Fanuc KAREL source: kt00486.KL

-- PROVISIONAL review KL for V770-1; original PC SHA256 9c85cafd3e05790770e6d16274b2af673c194925847be50b8fe71cd2a08aa8ed
-- Incomplete behavior may be omitted. Consult companion uncertainty JSON. Do not deploy.
PROGRAM KT00486
%NOLOCKGROUP
-- UNRESOLVED_DECL P1 type=000101
-- UNRESOLVED_DECL P2 type=000106
-- UNRESOLVED_DECL OUT type=000106
BEGIN
  -- UNRESOLVED_PC offsets 5-20; opcodes 2E,22,32,35
  -- UNRESOLVED_PC offsets 25-59; opcodes 49,49,7E,60,7E,4A
  -- UNRESOLVED_PC offsets 64-68; opcodes 7F
END KT00486
